{attribute 'qualified_only'}
{attribute 'strict'}
{attribute 'to_string'}
TYPE EDataFrame :
(
	_8N1 := 3,
	_8E1 := 4
);
END_TYPE

(* stored: Version 1.1.0.1, ProductVersion 3.1.4024.3
   DUT EDataFrame: Id {61404d4e-6602-4907-8d63-e9af39e80a53} *)
